TEXTLIST tlDevices
  0 = 'Bottle Sensor' | EN: 'Bottle Sensor' | PL: 'Bottle Sensor'
  1 = 'Bottle Eject Sensor' | EN: 'Bottle Eject Sensor' | PL: 'Bottle Eject Sensor'
  2 = 'Drawer Bottle Sensor' | EN: 'Drawer Bottle Sensor' | PL: 'Drawer Bottle Sensor'
  3 = 'Drawer Lock' | EN: 'Drawer Lock' | PL: 'Drawer Lock'
  4 = 'Weight' | EN: 'Weight' | PL: 'Weight'
  5 = 'Out Conveyor' | EN: 'Out Conveyor' | PL: 'Out Conveyor'
   = ''
END_TEXTLIST

(* stored: Version 1.1.0.1, ProductVersion 3.1.4024.15
   TextList tlDevices: Id {09652da2-fae6-49b9-9b2a-10e94f8e2354} *)
